{attribute addProperty BoxType "EK1122-0000-0018"}
{attribute addProperty Id "Beckhoff_ELM36xxsub_EK1100EK1100_179A0949162"}
{attribute addProperty CRC "3669837284"}
{attribute addProperty SizeInBites "16"}
{attribute addProperty SizeInBytes "2"}
TYPE Beckhoff_ELM36xxEK1122_DABD45E4 EXTENDS EK1122_179A0949 :
STRUCT
	{attribute addProperty Name "Beckhoff_ELM36xxsub_EK1100"}
	Beckhoff_ELM36xxsub_EK1100 : EK1100_179A0949;
END_STRUCT
END_TYPE

(* stored: Version 1.2.0.0, ProductVersion 3.1.4024.9
   DUT Beckhoff_ELM36xxEK1122_DABD45E4: Id {9e798b2e-5a3a-4db2-bdd9-849085fd7635} *)
